// TIA Portal V20 export
// export: Created 2025-12-01T14:57:44.1171093Z, ExportSetting None, DisplayName Totally Integrated Automation Portal, DisplayVersion V20 Update 3, DisplayName TIA Portal Openness, DisplayVersion V20 Update 3, DisplayName TIA Portal Version Control Interface, DisplayVersion V20 Update 3, DisplayName STEP 7 Professional, DisplayVersion V20 Update 3, DisplayName STEP 7 Safety, DisplayVersion V20 Update 2, DisplayName WinCC Basic/Comfort/Advanced, DisplayVersion V20 Update 3, DisplayName WinCC Professional, DisplayVersion V20 Update 3, DisplayName WinCC Unified, DisplayVersion V20 Update 3
FUNCTION "FC528_Form_Lec_Mod_SICK_PN_ALF" : Void   // FC528, STL
{ S7_Optimized_Access := 'FALSE' }
AUTHOR : ROUTER_A
NAME : 20181011
VERSION : 3.4
// stored: AutoNumber false
   VAR_INPUT
      Numero_Red : UInt;   // Red Actual de Lectura
      Datos_Red : "ROUT_Conf_Bucle_Lect_SCR";
   END_VAR
   VAR_IN_OUT
      CNT_LectCiclo : UInt;
   END_VAR
   VAR_TEMP
      Datos_E_Scanner : Array[0.."ROUT_Long_Dat_Scanner"] of Byte;
      EAB_Lectura : UInt;   // Byte 0 Entradas/Salidas del Scanner
      Datos_Diagnostico : Word;
      PunteroSCR_A : DWord;
      caracter_relleno : Char;
      retvalue : Int;
      Numero_Caracteres : UInt;
      CNT_Escritura : UInt;
      SCR_Actual : UInt;
      NumScanner : UInt;
      AUX_NumScanner : UInt;
      cero : Byte;
      CNT_Lectura : UInt;
      CNT_Datos_Pantalla : UInt;
   END_VAR
BEGIN

NETWORK
TITLE = Inicializar
// -- Calcular la dirección de lectura del scanner actual

      L     #Datos_Red.SCR_Actual;  // Direccion de E/S de Scanner
      L     #Datos_Red.NodoInicial;  // (Nodo * Long. Datos) + Address Incio
      -I;
      L     "ROUT_Long_Dat_Scanner";
      *I;
      L     #Datos_Red.AddresInicial;
      +I;
      T     #EAB_Lectura;

      L     0;
      T     #cero;


// ----------------------------------------------------------------------
// --- Calculo de Punteros   E / S

      L     #EAB_Lectura;  //--- Obtener Direccion entrada Scanner
      SLD   3;  //    Dar formato de Integer a Puntero
      L     P#3.0;  //--  EB_Lectura + 3 Byte
      +D;  //    Leer de PAB
      T     #PunteroSCR_A;

// -------------------------------------------------------------------------------------
// --- Numero de SCR Actual

      L     #Datos_Red.SCR_Actual;
      T     #SCR_Actual;


// -------------------------------------------------------------------------------------

// -------------------------------------------------------------------------------------
// obtener el caracter de relleno

      L     "ROUT_CaracterRelleno";
      T     #caracter_relleno;
// -------------------------------------------------------------------------------------


NETWORK
TITLE = Determinar Nueva Lectura
// -------------------------------------------------------------------------------------
// recogida de todos los datos del scanner

      CALL  "FC570_Leer_Zona_Entradas"
      ( Inicio_Zona := #EAB_Lectura,
        Long_Zona   := "ROUT_Long_Dat_Scanner",
        Datos_Zona  := #Datos_E_Scanner
      );

// Nieves: hay que revisar en un funcionamiento con scanner real
//  como quedan los datos de diagnóstico


      L     #Datos_E_Scanner[0];
      T     #Datos_Diagnostico.%B0;
      L     #Datos_E_Scanner[1];
      T     #Datos_Diagnostico.%B1;


// -------------------------------------------------------------------------------------
// ---  pasamos a ver el telegrama del scanner
// --- Comprobamos si hay Nueva Lectura de Scanner
// --- si el número de lectura disponible es igual a la ultima tratada
// --- Significa que no hay ninguna nueva lectura pendiente de ser tratada


      L     "DB214_CNT_Mens_SCR".RedScanners[#Numero_Red].CNT_NODO_PROF_SCR[#SCR_Actual];  // --- Memoria con el número de la ultima lectura tratada
      L     #Datos_E_Scanner[3];  // --- Numero de lectura disponible para ser tratada
      ==I;
      JC    Fin_funcion;

// -------------------------------------------------------------------------------------


NETWORK
TITLE = Obtener Identificador Scanner (modif a 3digit el 27/08/18)

// -------------------------------------------------------------------------------------
// --- Numero de Numero del Scanner
      L     #Datos_E_Scanner[7];  // --- Obtener Centenas
      L     W#16#F;  //     Eliminamos la parte alta del BYTE
      AW;  //     Multiplicamos por el peso del caracter
      L     100;
      *I;
      T     #AUX_NumScanner;  // --- Lo Paso al valor del NODO

      L     #Datos_E_Scanner[8];  // --- Obtener Decenas
      L     W#16#F;  //     Eliminamos la parte alta del BYTE
      AW;  //     Multiplicamos por el peso del caracter
      L     10;
      *I;
      L     #AUX_NumScanner;  // --- Lo sumamo al valor del NODO
      +I;
      T     #AUX_NumScanner;  // --- Lo sumamo al valor del NODO


      L     #Datos_E_Scanner[9];  // --- Obtener Unidad
      L     W#16#F;  //     Eliminamos la parte alta del BYTE
      AW;  //     Multiplicamos por el peso del caracter
      L     1;
      *I;
      L     #AUX_NumScanner;  // --- Lo sumamo al valor del NODO
      +I;
      T     #NumScanner;  // --- Lo sumamo al valor del NODO

// -------------------------------------------------------------------------------------
// -- si el numero del scanner es 0, ha habido algún problema NIEVES PENDIENTE DEFINIR

      SET;
      L     #NumScanner;  // -- Descartar cualquier lectura de identificadores de scanner 0
      L     0;
      ==I;
      JC    Fin_Bucle;

// -------------------------------------------------------------------------------------


NETWORK
TITLE = Validar Escritura en DB e inicar Registros
// -------------------------------------------------------------------------------------
// --- Comprobacion de nuemro de caracteres leidos

      L     "ROUT_Long_Etiqueta";  // --- Carga Dato de Número de caracteres de etiquetas esperados en el DB
      L     4;  // -- le añadimos 4 porque los 4 digitos qu emanda de identificador nos se guardan realmente pero se cuentan en el mensaje.
      +I;
      L     #Datos_E_Scanner[5];  // --- Carga el dato de Número de caracteres Leidos
      -I;
      T     #Numero_Caracteres;  // --- Posición donde empezar a escribir la etiqueta en DB

      SET;
      L     #Numero_Caracteres;
      L     0;
      <=I;
      JC    Error_lectura;  // --- Si resultado <=0 LONGITUD LECTURA de scanner FUERA DE RANGO


// -------------------------------------------------------------------------------------
// --- Validar si se puede leer la nueva lectura
// --- la condición es que la lectura anterior esté tratada

      SET;
      L     "DB211_Lecturas_Scanner".Lec_Scanner[#NumScanner].Lectura_SCR[0];
      L     'N';  //      Carga el caracter 'N' para compara
      ==I;  //      Si es igual no tratamos la lectura actual
      JC    Fin_funcion;  //      ESPERAMOS QUE SE TRATE LA LECTURA ANTERIOR

// -------------------------------------------------------------------------------------


NETWORK
TITLE = Formatear Lectura Correcta de Escanner
// -------------------------------------------------------------------------------------
// --- Incializalizamoms la lectura

      CALL  FILL
      ( BVAL    := #cero,
        RET_VAL := #retvalue,
        BLK     := "DB211_Lecturas_Scanner".Lec_Scanner[#NumScanner]
      );

      CALL  FILL
      ( BVAL    := #cero,
        RET_VAL := #retvalue,
        BLK     := "DB905_Estado_Escaners".Escaner[#NumScanner].Lectura
      );


      L     1;
      T     #CNT_Escritura;  // --- Inicializa el contador de caracteres de escritura
      L     11;
      T     #CNT_Lectura;
      L     0;
      T     #CNT_Datos_Pantalla;



      L     'N';
      T     "DB211_Lecturas_Scanner".Lec_Scanner[#NumScanner].Lectura_SCR[0];  //      Carga el primer caracter de la etiqueta existente



// -------------------------------------------------------------------------------------
// --- Bucle de lectura de Etiqueta

Inicio_bucle:NOP   0;  // --- INICIO BUCLE ETIQUETA
      L     #CNT_Escritura;
      L     #Numero_Caracteres;  //     Si estamos a la izquierda del primer Caracter ponemos la 'N'
      >=I;
      JC    Escribir_Etiqueta;  // --- Tomamos caracter de lectura de escaner ?


      L     #caracter_relleno;  // Nieves: modificación para que el JDT pueda truncar la lectura más facilmente   20/09/16
      T     "DB211_Lecturas_Scanner".Lec_Scanner[#NumScanner].Lectura_SCR[#CNT_Escritura];
      T     "DB905_Estado_Escaners".Escaner[#NumScanner].Lectura[#CNT_Datos_Pantalla];  // transfiero tambien al array temporal que nos hemos creado

      L     1;  // --- Incrementa contador caracteres
      L     #CNT_Datos_Pantalla;
      +I;
      T     #CNT_Datos_Pantalla;

      L     1;  // --- Incrementa contador caracteres
      L     #CNT_Escritura;
      +I;
      T     #CNT_Escritura;


// comprobación del caracter de escritura para no salirnos de rango
      SET;
      L     #CNT_Escritura;  // --- Mirar si se ha acabo la etiqueta
      L     "ROUT_Long_Etiqueta";
      <I;  // --- Si no llegamos al final repetimos el bucle
      JC    Inicio_bucle;

// si no hemos saltado es que hemos llegado al último caracter de escritura y tenemos que salir

      JU    Fin_Bucle;


// -------------------------------------------------------------------------------------
// -- Escribimos ahora la etiqueta

Escribir_Etiqueta:NOP   0;
      L     #Datos_E_Scanner[#CNT_Lectura];  // --- Leer carcater de la Etiqueta
      T     "DB211_Lecturas_Scanner".Lec_Scanner[#NumScanner].Lectura_SCR[#CNT_Escritura];  //     escribirlo en el registro de la etiqueta
      T     "DB905_Estado_Escaners".Escaner[#NumScanner].Lectura[#CNT_Datos_Pantalla];  // transfiero tambien al array temporal que nos hemos creado



// -------------------------------------------------------------------------------------
// -- incrementamos los contadores para pasar al siguiente caracter
siguiente_caracter:NOP   0;

      L     1;  // --- Incrementa contador caracteres
      L     #CNT_Escritura;
      +I;
      T     #CNT_Escritura;

      L     1;  // --- Incrementa contador caracteres
      L     #CNT_Lectura;
      +I;
      T     #CNT_Lectura;

      L     1;  // --- Incrementa contador caracteres
      L     #CNT_Datos_Pantalla;
      +I;
      T     #CNT_Datos_Pantalla;


      L     #CNT_Escritura;  // --- Mirar si se ha acabo la etiqueta
      L     "ROUT_Long_Etiqueta";
      <I;  // --- Si no llegamos al final repetimos el bucle
      JC    Inicio_bucle;

      JU    Fin_Bucle;  // --- Si termina la lectura correctamente cerramos protocolo



NETWORK
TITLE = Error lectura etiqueta no esperada
// -------------------------------------------------------------------------------------
// ---  Rellenar de error de etiqueta --> 'N000000000'

Error_lectura:NOP   0;

      L     1;  // --- Incializar CNT de Caracteres Escritos
      T     #CNT_Escritura;
      L     0;
      T     #CNT_Datos_Pantalla;


      L     'N';  // --- Caracter 'N'
      T     "DB211_Lecturas_Scanner".Lec_Scanner[#NumScanner].Lectura_SCR[0];


bucle_error:NOP   0;

      L     '0';  // --- Caracter '0'
      T     "DB211_Lecturas_Scanner".Lec_Scanner[#NumScanner].Lectura_SCR[#CNT_Escritura];
      T     "DB905_Estado_Escaners".Escaner[#NumScanner].Lectura[#CNT_Datos_Pantalla];


// -- incrementamos los contadores para desplazarnos en la estructura

      L     1;  // --- Incrementa contador caracteres
      L     #CNT_Escritura;
      +I;
      T     #CNT_Escritura;

      L     1;  // --- Incrementa contador caracteres
      L     #CNT_Datos_Pantalla;
      +I;
      T     #CNT_Datos_Pantalla;


      L     #CNT_Escritura;  // --- Mirar si se ha acabo la etiqueta
      L     "ROUT_Long_Etiqueta";
      <I;  // --- Si no llegamos al final repetimos el bucle ?
      JC    bucle_error;

      JU    Fin_Bucle;  // --- Si termina la lectura correctamente cerramos protocolo



NETWORK
TITLE = Confirmar al Scanner de leida la etiqueta
// -------------------------------------------------------------------------------------
// --- Confirmar al Scanner de leida la etiqueta

Fin_Bucle:NOP   0;

// -- Guardamos los datos de la etiqueta recogida en el DB

      L     #Datos_E_Scanner[3];  // --- Obtenemos un puntero al número de telegrama del Scanner
      T     QB [#PunteroSCR_A];  // --- Confirmamos la lectura con el número de telegrama del Scanner

      L     #Datos_E_Scanner[3];  // --- La lectura ha sido tratada anteriormente
      T     "DB214_CNT_Mens_SCR".RedScanners[#Numero_Red].CNT_NODO_PROF_SCR[#SCR_Actual];  //     Guardar el ID de la recepción y en el envio


      L     #CNT_LectCiclo;  // --- Incrementa el Numero de lecturas por ciclo
      L     1;
      +I;
      T     #CNT_LectCiclo;


NETWORK
TITLE = Actualizar datos pantalla
//===============================================================================================
//-- volcamos el dato del diagnóstico

      CALL  BLKMOV
      ( SRCBLK  := #Datos_Diagnostico,
        RET_VAL := #retvalue,
        DSTBLK  := "DB905_Estado_Escaners".Escaner[#NumScanner].Diagnostico
      );



//===============================================================================================


NETWORK
TITLE = salir de la funcion
// -------------------------------------------------------------------------------------
// --- Se sale de la función

Fin_funcion:NOP   0;

END_FUNCTION
